// TIA Portal V20 export
VAR_GLOBAL   // PLC tag table "LAcycCom_Drives"
END_VAR
